DATA_BLOCK "DB"
{ S7_Optimized_Access := 'false' }
    VAR
        aut_r: REAL;
        aut_b: BOOL;
        aut_i: DINT;
        aut_tii: TupleStruct2;
        aut: BOOL;
        inp: REAL;
        c: REAL;
        preset_c: TIME;
        firstRun: BOOL;
    END_VAR
BEGIN
    firstRun := TRUE;
END_DATA_BLOCK
